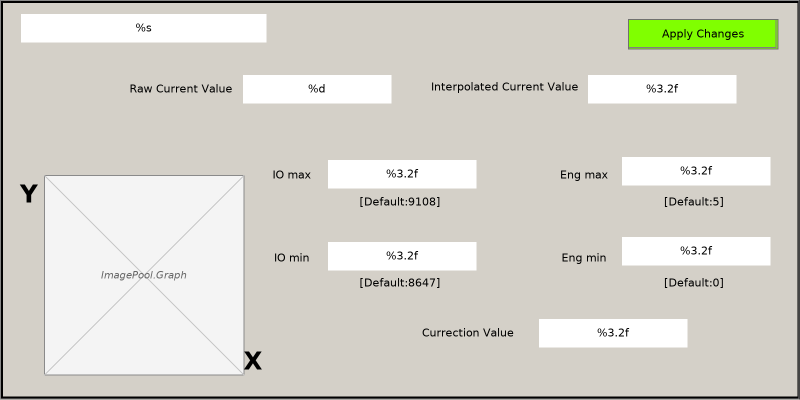
VISUALIZATION vSensorCalibrate_1_2  // 800x400
VAR_IN_OUT
	vAnalogSensor:FB_AnalogSensor;
END_VAR
    Rectangle (0,0 800x399)
    Image (44,175 200x200), image: ImagePool.Graph
    Label (228,346 50x30), "X"
    Label (4,179 50x30), "Y"
    Label (106,74 150x30), "Raw Current Value"
    Textfield (621,156 150x30), "%3.2f", text variable: vAnalogSensor.EngMax
        OnMouseClick: write the text variable via Default
    Textfield (621,236 150x30), "%3.2f", text variable: vAnalogSensor.EngMin
        OnMouseClick: write the text variable via Default
    Textfield (327,159 150x30), "%3.2f", text variable: vAnalogSensor.IoMax
        OnMouseClick: write the text variable via Default
    Textfield (327,241 150x30), "%3.2f", text variable: vAnalogSensor.IoMin
        OnMouseClick: write the text variable via Default
    Textfield (242,74 150x30), "%d", text variable: vAnalogSensor.iAnalogIn
    Label (430,72 150x30), "Interpolated Current Value"
    Textfield (587,74 150x30), "%3.2f", text variable: vAnalogSensor.rSensorVal
    Button (628,19 150x30), "Apply Changes"
        OnMouseClick: execute { MAIN.bSetPerData:=true; }
    Label (393,318 150x30), "Currection Value"
    Textfield (538,318 150x30), "%3.2f", text variable: vAnalogSensor.rCorrection
        OnMouseClick: write the text variable via Default
    Textfield (20,13 247x30), "%s", text variable: vAnalogSensor.sSensorName
    Label (217,160 150x30), "IO max"
    Label (217,243 150x30), "IO min"
    Label (509,160 150x30), "Eng max"
    Label (509,243 150x30), "Eng min"
    Label (325,187 150x30), "[Default:9108]"
    Label (619,187 150x30), "[Default:5]"
    Label (325,268 150x30), "[Default:8647]"
    Label (619,268 150x30), "[Default:0]"
END_VISUALIZATION

(* stored: Version 1.1.0.1, ProductVersion 3.1.4024.12
   Visu vSensorCalibrate_1_2: Id {d216569b-1318-46db-b323-a7658e07bbed} *)
